Fanuc TP program (LS listing): PRG.LS

/PROG  PRG
/ATTR
OWNER		= MNEDITOR;
COMMENT		= "";
PROG_SIZE	= 227;
CREATE		= DATE 21-04-07  TIME 13:40:18;
MODIFIED	= DATE 21-04-09  TIME 11:28:38;
FILE_NAME	= ;
VERSION		= 0;
LINE_COUNT	= 1;
MEMORY_SIZE	= 595;
PROTECT		= READ_WRITE;
TCD:  STACK_SIZE	= 0,
      TASK_PRIORITY	= 50,
      TIME_SLICE	= 0,
      BUSY_LAMP_OFF	= 0,
      ABORT_REQUEST	= 0,
      PAUSE_REQUEST	= 0;
DEFAULT_GROUP	= 1,*,*,*,*;
CONTROL_CODE	= 00000000 00000000;
/APPL
/APPL

AUTO_SINGULARITY_HEADER;
  ENABLE_SINGULARITY_AVOIDANCE   : TRUE;

  AUTOZONE_INTERFERENCE_AVOID;
    AUTOZONE_ENABLED         : FALSE;
    AUTOZONE_SCHEDULE_NUMBER : 1;
/MN
   1:  R[164]=(R[163]-((R[163] DIV 99)*198)) ;
/POS
/END
